FUNCTION F_ITC_SendRDR : BOOL
(**************************************************************************************
 * 	Application		:	BoxControl Framework
 *	Revision		:	$Revision: 404529 $
 *	Revision date	:	$Date: 2018-04-23 08:21:38 +0200 (Mo., 23 Apr 2018) $
 *	Last changed by	:	$Author: b7bolm $
 *	URL				:	$URL: http://almscdc.swisslog.com/repo/SWPD/Development/BoxControlFramework/20_Release/trunk/01_Software/BCF/BCF/JumpStart/20_Product/10_App/11_Com/10_Lib/10_Conv/11_ITC/F_ITC_SendRDR.TcPOU $
 *
 *	Purpose			:	Wrap message - RDR
 *
 * ------------------------------------------------------------------------------------
 *	Copyright Swisslog [IP AG], Switzerland. All rights reserved.
 * 
 * ------------------------------------------------------------------------------------
 *	
 * 	Revision History: 
 *
 * 	VERSION			DATE			INITIALS			DESCRIPTION
 *	0.1				01.01.2001		swl					Example
 *
 **************************************************************************************)
VAR_INPUT
	eChannelSrc			: E_MFCS_Channel; // Source communicaton channel
	PositionName		: STRING(Conveyor.POSITION_STRINGLENGTH); // SIS MM-GGG-EEEE-FF-Z
	CommandDataIndex	: DINT;
	AssignmentID		: UDINT; // assignment id
	GroupID				: ULINT;
	eReturnCode			: E_ErrorConv; // Return code
END_VAR
VAR
	RDR				: ST_ITC_RDR; 
END_VAR

// Map values
RDR.Position := PositionName;
RDR.CommandDataIndex := CommandDataIndex;
RDR.AssignmentID := AssignmentID;
RDR.GroupID := GroupID;
RDR.ReturnCode := eReturnCode;

// Forward to ITC
F_ITC_SendRDR := fbITC_Manager.M_SendData(
					meChannel	:= eChannelSrc,
					mMsgType	:= E_ITC_MsgTypeConv.ROBOT_DELETE_REPORT,
					mpData		:= ADR(RDR),
					mLen		:= SIZEOF(RDR));

END_FUNCTION

(* stored: Version 1.1.0.1, ProductVersion 3.1.4022.12
   POU F_ITC_SendRDR: Id {883a4f2d-31ff-4d84-8e8c-af124db74b81}, SpecialFunc None *)
